// TwinCAT 3 PLC project Main_Code
// ProgramVersion: 3.1.4026.14
// libraries:
//   Tc2_Standard, * (Beckhoff Automation GmbH)
//   Tc2_System, * (Beckhoff Automation GmbH)
//   Tc3_Database, * (Beckhoff Automation GmbH)
// project tree:
//   DUTs/ DUT_SQL.TcDUT
//   / PlcTask.TcTTO
//   POUs/ FC_SQL_InsertCommands_TempSensor.TcPOU, MAIN.TcPOU, FC_SQL_InsertCommands_LoadCell.TcPOU, FC_SQL_InsertCommands_Encoder.TcPOU
// real-time tasks:
//   TASK PlcTask: cycle T#1ms, priority 20, ADS port 350
// I/O:
//   DEVICE Device 1 (EtherCAT), AmsNetId 145.44.56.216.2.1

CONFIGURATION Main_Code
    RESOURCE PLC ON TwinCAT3
        TASK PlcTask(INTERVAL := T#1ms, PRIORITY := 20);
        PROGRAM MAIN WITH PlcTask : MAIN;
    END_RESOURCE
END_CONFIGURATION

// ---- DUTs/DUT_SQL.TcDUT
TYPE DUT_SQL :
STRUCT
    SensorValue : INT;
    SampleNr : INT;
    Timestamp : STRING(50);
END_STRUCT
END_TYPE

// ---- POUs/MAIN.TcPOU
PROGRAM MAIN
VAR
    FB_SQLDatabaseEvt : FB_SQLDatabaseEvt(sNetID := '', tTimeout := T#5S);
    FB_SQLCommandEvt  : FB_SQLCommandEvt(sNetID := '', tTimeout := T#5S);
    FB_SQLResultEvt   : FB_SQLResultEvt(sNetID := '', tTimeout := T#5S);

    iStep: INT;
    SQL_Commands: ARRAY[1..2] OF STRING(255);
    iSampleNr: INT := 1;
    iLoadCellValue AT %I*: INT;
	iLoadCellPreviousValue : INT;
	iTempSensorValue AT %I*: INT;
	iEncoderValue AT %I*: INT;

    sSelectDataCommand : STRING(255);
END_VAR


CASE iStep OF
    0:
        iStep := 10;

    10: // Connect to Database
        FB_SQLDatabaseEvt.Connect(hDBID := 1);
        IF FB_SQLDatabaseEvt.bConnected THEN
            iStep := 20;
        END_IF

    20: // Create SQL Command Object
        FB_SQLDatabaseEvt.CreateCmd(pSQLCommand := ADR(FB_SQLCommandEvt));
        IF NOT FB_SQLDatabaseEvt.bBusy THEN
            iStep := 30;
        END_IF

    30: // Generate INSERT Commands
		SQL_Commands[1] := FC_SQL_InsertCommands_Encoder(iEncoderValue, iSampleNr);
		SQL_Commands[1] := FC_SQL_InsertCommands_TempSensor(iTempSensorValue, iSampleNr);
        //check if loadcell value changed
		IF ABS(iLoadCellValue - iLoadCellPreviousValue) > 100 THEN
			SQL_Commands[1] := FC_SQL_InsertCommands_LoadCell(iLoadCellValue, iSampleNr);
    		iSampleNr := iSampleNr + 1; // Increment sample number
    		iLoadCellPreviousValue := iLoadCellValue; // Update previous value tracker
		END_IF
		 iStep := 40;

    40: // Execute Insert Command
        IF FB_SQLCommandEvt.Execute(pSQLCmd := ADR(SQL_Commands[1]), cbSQLCmd := SIZEOF(SQL_Commands[1])) THEN
            iStep := 50;
        END_IF

    50: // Prepare SELECT Query
        sSelectDataCommand := 'SELECT TOP 10 * FROM [db_accessadmin].[TempSensor_Data] ORDER BY Time DESC;';
        iStep := 60;

    60: // Execute SELECT Command
         FB_SQLCommandEvt.ExecuteDataReturn(
            pSQLCmd := ADR(sSelectDataCommand),
            cbSQLCmd := SIZEOF(sSelectDataCommand),
            pSQLDBResult := ADR(FB_SQLResultEvt)); 
        iStep := 30;
   

END_CASE

END_PROGRAM

// ---- POUs/FC_SQL_InsertCommands_Encoder.TcPOU
FUNCTION FC_SQL_InsertCommands_Encoder : STRING(255)
VAR_INPUT
    iSensorValue: INT;
    iSampleNr: INT;
END_VAR

FC_SQL_InsertCommands_Encoder := 'INSERT INTO [db_accessadmin].[Encoder] (SensorValue, SampleNr, Time) VALUES (';
FC_SQL_InsertCommands_Encoder := CONCAT(FC_SQL_InsertCommands_Encoder, INT_TO_STRING(iSensorValue));
FC_SQL_InsertCommands_Encoder := CONCAT(FC_SQL_InsertCommands_Encoder, ', ');
FC_SQL_InsertCommands_Encoder := CONCAT(FC_SQL_InsertCommands_Encoder, INT_TO_STRING(iSampleNr));
FC_SQL_InsertCommands_Encoder := CONCAT(FC_SQL_InsertCommands_Encoder, ', GETDATE());');

END_FUNCTION

// ---- POUs/FC_SQL_InsertCommands_TempSensor.TcPOU
FUNCTION FC_SQL_InsertCommands_TempSensor : STRING(255)
VAR_INPUT
    iSensorValue: STRING;
    iSampleNr: INT;
	iSensorID: INT;
END_VAR

FC_SQL_InsertCommands_TempSensor := 'INSERT INTO [db_accessadmin].[TempSensor] (SensorValue, SampleNr, Time, SensorID) VALUES (';
FC_SQL_InsertCommands_TempSensor := CONCAT(FC_SQL_InsertCommands_TempSensor, iSensorValue);
FC_SQL_InsertCommands_TempSensor := CONCAT(FC_SQL_InsertCommands_TempSensor, ', ');
FC_SQL_InsertCommands_TempSensor := CONCAT(FC_SQL_InsertCommands_TempSensor, INT_TO_STRING(iSampleNr));
FC_SQL_InsertCommands_TempSensor := CONCAT(FC_SQL_InsertCommands_TempSensor, ', GETDATE(), ');
FC_SQL_InsertCommands_TempSensor := CONCAT(FC_SQL_InsertCommands_TempSensor, INT_TO_STRING(iSensorID));
FC_SQL_InsertCommands_TempSensor := CONCAT(FC_SQL_InsertCommands_TempSensor, ');');

END_FUNCTION

// ---- POUs/FC_SQL_InsertCommands_LoadCell.TcPOU
FUNCTION FC_SQL_InsertCommands_LoadCell : STRING(255)
VAR_INPUT
    iSensorValue: INT;
    iSampleNr: INT;
END_VAR

FC_SQL_InsertCommands_LoadCell := 'INSERT INTO [db_accessadmin].[LoadCell] (SensorValue, SampleNr, Time) VALUES (';
FC_SQL_InsertCommands_LoadCell := CONCAT(FC_SQL_InsertCommands_LoadCell, INT_TO_STRING(iSensorValue));
FC_SQL_InsertCommands_LoadCell := CONCAT(FC_SQL_InsertCommands_LoadCell, ', ');
FC_SQL_InsertCommands_LoadCell := CONCAT(FC_SQL_InsertCommands_LoadCell, INT_TO_STRING(iSampleNr));
FC_SQL_InsertCommands_LoadCell := CONCAT(FC_SQL_InsertCommands_LoadCell, ', GETDATE());');

END_FUNCTION
